FUNCTION_BLOCK TEST_NEB (* Test NE function on bit strings *)
  (* Standard: 61499-1 *)
  (* Version 0.0, 2006-09-14, JHC, Holobloc Inc *)
  (* Compiler header: package fb.rt.test; *)
  (* Compiler classdef: SimpleFB *)
  (* Compiler Java Sun JDK 1.5.0 *)
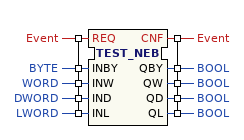
  EVENT_INPUT
    REQ WITH INBY, INW, IND, INL; (* Normal Execution Request *)
  END_EVENT
  EVENT_OUTPUT
    CNF WITH QBY, QW, QD, QL; (* Execution Confirmation *)
  END_EVENT
  VAR_INPUT
    INBY : BYTE;
    INW : WORD;
    IND : DWORD;
    INL : LWORD;
  END_VAR
  VAR_OUTPUT
    QBY : BOOL;
    QW : BOOL;
    QD : BOOL;
    QL : BOOL;
  END_VAR
  ALGORITHM REQ IN FBD:
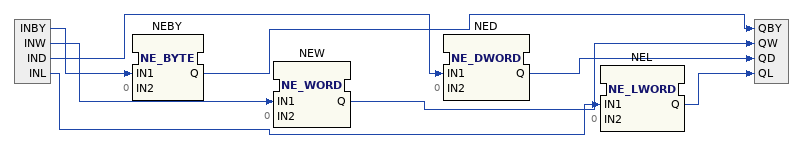
    FBS
      NEBY : NE_BYTE(IN2 := 0);
      NEW : NE_WORD(IN2 := 0);
      NED : NE_DWORD(IN2 := 0);
      NEL : NE_LWORD(IN2 := 0);
    END_FBS
    DATA_CONNECTIONS
      INBY TO NEBY.IN1;
      NEBY.Q TO QBY;
      INW TO NEW.IN1;
      NEW.Q TO QW;
      IND TO NED.IN1;
      NED.Q TO QD;
      INL TO NEL.IN1;
      NEL.Q TO QL;
    END_CONNECTIONS
  END_ALGORITHM
END_FUNCTION_BLOCK
